FUNCTION_BLOCK ASR_AX_SERVER_0_CLIENT_1_0 (* Receive 2 independent remote OPC-UA method calls via SERVER_0 (Set/Reset) and write the resulting state back via CLIENT_1_0, driven by an ASR_AX bidirectional adapter Plug *)
  (* Standard: 61499-2; Description: Copyright (c) 2026 HR Agrartechnik GmbH This program and the accompanying materials are made available under the terms of the Eclipse Public License 2.0 which is available at https://www.eclipse.org/legal/epl-2.0/ SPDX-License-Identifier: EPL-2.0 *)
  (* Version 1.0, 2026-09-03, Franz Höpfinger, HR Agrartechnik GmbH, initial API and implementation and/or initial documentation *)
  PACKAGE adapter::net;
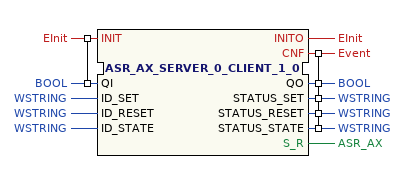
  EVENT_INPUT
    INIT : EInit WITH QI; (* Initialization *)
  END_EVENT
  EVENT_OUTPUT
    INITO : EInit; (* Initialization Confirm *)
    CNF WITH QO, STATUS_SET, STATUS_RESET, STATUS_STATE; (* QO/STATUS updated *)
  END_EVENT
  VAR_INPUT
    QI : BOOL;
    ID_SET : WSTRING; (* Lokale Methodenadresse (ACTION=CREATE_METHOD) fuer den Set-Methodenaufruf *)
    ID_RESET : WSTRING; (* Lokale Methodenadresse (ACTION=CREATE_METHOD) fuer den Reset-Methodenaufruf *)
    ID_STATE : WSTRING; (* Remote-Ziel-Adresse (ACTION=WRITE) fuer den Zustand *)
  END_VAR
  VAR_OUTPUT
    QO : BOOL; (* TRUE nur wenn SET_SERVER, RESET_SERVER und STATE_CLIENT aktuell alle QO=TRUE melden *)
    STATUS_SET : WSTRING; (* STATUS von SET_SERVER *)
    STATUS_RESET : WSTRING; (* STATUS von RESET_SERVER *)
    STATUS_STATE : WSTRING; (* STATUS von STATE_CLIENT *)
  END_VAR
  PLUGS
    S_R : adapter::types::bidirectional::ASR_AX; (* Set/Reset (in), Zustand (out) *)
  END_PLUGS
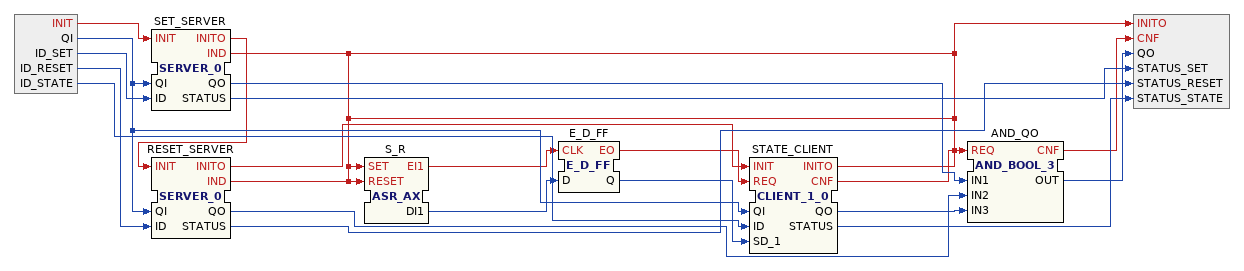
  FBS
    SET_SERVER : iec61499::net::SERVER_0;
    RESET_SERVER : iec61499::net::SERVER_0;
    E_D_FF : iec61499::events::E_D_FF;
    STATE_CLIENT : iec61499::net::CLIENT_1_0;
    AND_QO : iec61131::booleanOperators::AND_BOOL_3;
  END_FBS
  EVENT_CONNECTIONS
    INIT TO SET_SERVER.INIT;
    SET_SERVER.INITO TO RESET_SERVER.INIT;
    RESET_SERVER.INITO TO STATE_CLIENT.INIT;
    STATE_CLIENT.INITO TO INITO;
    STATE_CLIENT.INITO TO AND_QO.REQ;
    SET_SERVER.IND TO S_R.SET;
    RESET_SERVER.IND TO S_R.RESET;
    S_R.EI1 TO E_D_FF.CLK;
    E_D_FF.EO TO STATE_CLIENT.REQ;
    SET_SERVER.IND TO AND_QO.REQ;
    RESET_SERVER.IND TO AND_QO.REQ;
    STATE_CLIENT.CNF TO AND_QO.REQ;
    AND_QO.CNF TO CNF;
  END_CONNECTIONS
  DATA_CONNECTIONS
    QI TO SET_SERVER.QI;
    QI TO RESET_SERVER.QI;
    QI TO STATE_CLIENT.QI;
    ID_SET TO SET_SERVER.ID;
    ID_RESET TO RESET_SERVER.ID;
    ID_STATE TO STATE_CLIENT.ID;
    S_R.DI1 TO E_D_FF.D;
    E_D_FF.Q TO STATE_CLIENT.SD_1;
    SET_SERVER.QO TO AND_QO.IN1;
    RESET_SERVER.QO TO AND_QO.IN2;
    STATE_CLIENT.QO TO AND_QO.IN3;
    AND_QO.OUT TO QO;
    SET_SERVER.STATUS TO STATUS_SET;
    RESET_SERVER.STATUS TO STATUS_RESET;
    STATE_CLIENT.STATUS TO STATUS_STATE;
  END_CONNECTIONS
END_FUNCTION_BLOCK
